// TIA Portal V19 export
TYPE "array2Months"
   STRUCT
      Current : Array[1.."MAX_DAYS_IN_MONTH"] of Real;
      Last : Array[1.."MAX_DAYS_IN_MONTH"] of Real;
   END_STRUCT;
END_TYPE
